PROGRAM MAIN
VAR
	x: LREAL;
	y: LREAL;
	z: LREAL;
END_VAR

END_PROGRAM

(* stored: Version 1.1.0.1, ProductVersion 3.1.4024.2
   POU MAIN: Id {1845b391-745b-40f8-973d-4ad23fa36772}, SpecialFunc None *)
